FUNCTION_BLOCK FB_925
VAR_INPUT
END_VAR
VAR_OUTPUT
END_VAR
VAR_IN_OUT
	VG	: ST_VG;
END_VAR
VAR
	rV : REAL;
	fbGaugeState : FB_PressureState;
	rMaxPressure	:	REAL := 760; //Torr
	rMinPressure	:	REAL := 1E-5; //Torr
END_VAR

(* Standard MKS 9XX series conversion *)
(* works for 972 and 925 *)

//Default setpoint 50 mT
IF VG.rVAC_SP = 0 THEN
	VG.rVAC_SP := 5E-2;
END_IF

rV := 10*INT_TO_REAL(VG.iPRESS_R)/32767;

IF rV >= 0.99 THEN
	IF rV >= 0.99 AND rV < 1 THEN
		VG.rPRESS := 1E-5;
	ELSE
		VG.rPRESS := LREAL_TO_REAL(EXPT(10, REAL_TO_LREAL(rV-6)));
	END_IF
	VG.xPRESS_OK := TRUE; //Backwards compatibility
ELSE
	VG.xPRESS_OK := FALSE;
END_IF

(* Pressure OK check *)
fbGaugeState.i_rV := rV;
fbGaugeState.i_MaxPressure := rMaxPressure;
fbGaugeState.i_MinPressure := rMinPressure;
fbGaugeState(iq_stVG:=VG);

(* Setpoint evaluation *)
VG.xAT_VAC := VG.xPRESS_OK AND (VG.rPRESS < VG.rVAC_SP);

END_FUNCTION_BLOCK

(* stored: Version 1.1.0.1, ProductVersion 3.1.4022.18
   POU FB_925: Id {2b25be69-d890-49a3-9eed-41a1523a8d75}, SpecialFunc None *)
